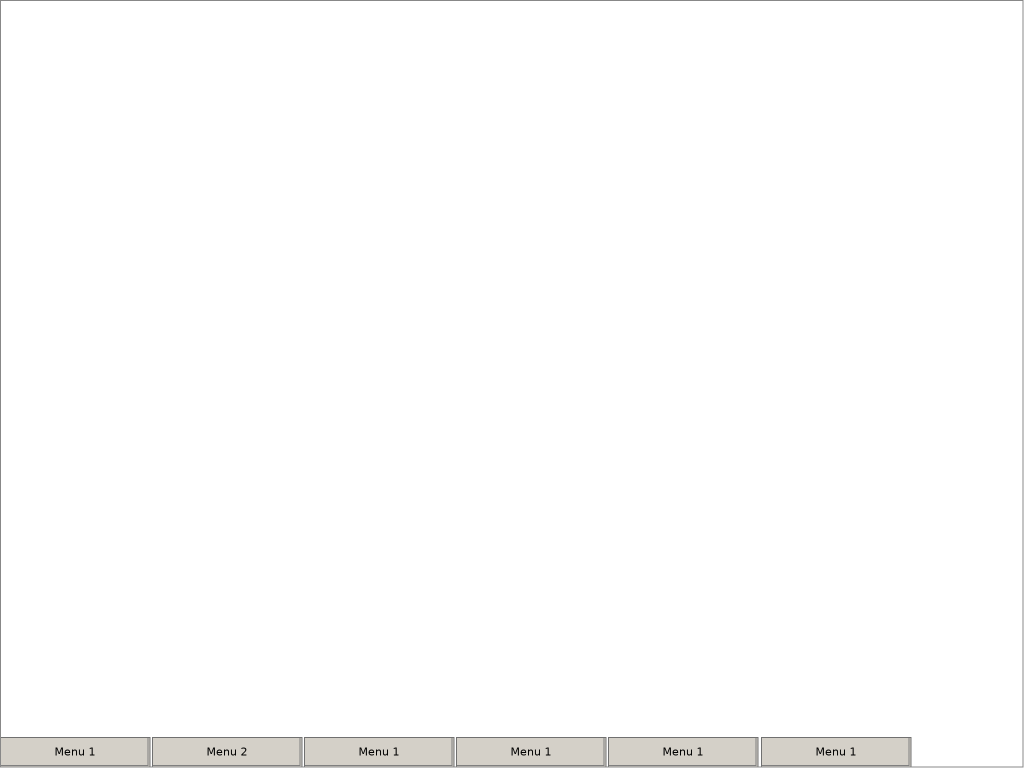
VISUALIZATION popup_test  // 1024x768
    Button (0,737 150x30), "Menu 1"
        OnMouseClick: OpenDialog Dialog=PopupMenu1, OpenModal=True, OpenCentered=True
    Button (159,789 2x1)
    Button (152,737 150x30), "Menu 2"
        OnMouseClick: OpenDialog Dialog=PopupMenu2, OpenModal=True, OpenCentered=True
    Button (304,737 150x30), "Menu 1"
        OnMouseClick: OpenDialog Dialog=PopupMenu1, OpenModal=True, OpenCentered=True
    Button (456,737 150x30), "Menu 1"
        OnMouseClick: OpenDialog Dialog=PopupMenu1, OpenModal=True, OpenCentered=True
    Button (608,737 150x30), "Menu 1"
        OnMouseClick: OpenDialog Dialog=PopupMenu1, OpenModal=True, OpenCentered=True
    Button (761,737 150x30), "Menu 1"
        OnMouseClick: OpenDialog Dialog=PopupMenu1, OpenModal=True, OpenCentered=True
END_VISUALIZATION

(* stored: Version 1.1.0.1, ProductVersion 3.1.4024.11
   Visu popup_test: Id {eab8c03a-eca7-08f1-3809-6df63cfd4c11} *)
